% RSLogix 500 project Car Parking System Using Counters.RSS, saved by version 8.30.00.16 %
PROJECT "UNTITLED"    % processor: Bul.1763 MicroLogix 1100 Series B %

PROGRAM FILES
  LAD 2   6 rungs

DATA FILES
  O0 OUTPUT  4 elements
  I1 INPUT  6 elements
  S2 STATUS  66 elements
  B3 BINARY  1 elements
  T4 TIMER  1 elements
  C5 COUNTER  1 elements
  R6 CONTROL  1 elements
  N7 INTEGER  1 elements
  F8 FLOAT  1 elements

LADDER 2
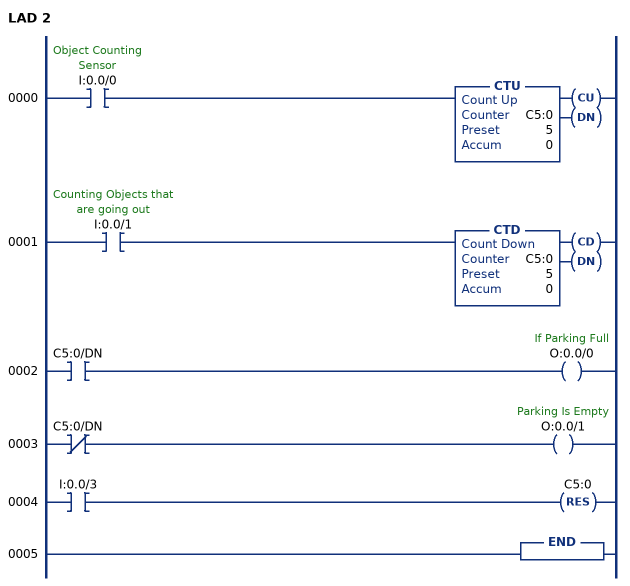
% Rung: 0 %
SOR XIC I:0.0/0 CTU C5:0 5 0 EOR
%   I:0.0/0  "Object Counting Sensor" %
% Rung: 1 %
SOR XIC I:0.0/1 CTD C5:0 5 0 EOR
%   I:0.0/1  "Counting Objects that are going out" %
% Rung: 2 %
SOR XIC C5:0/DN OTE O:0.0/0 EOR
%   O:0.0/0  "If Parking Full" %
% Rung: 3 %
SOR XIO C5:0/DN OTE O:0.0/1 EOR
%   O:0.0/1  "Parking Is Empty" %
% Rung: 4 %
SOR XIC I:0.0/3 RES C5:0 EOR
% Rung: 5 %
SOR END EOR

DATA TABLE (non-zero values as saved)
DATA C5
% .PRE .ACC %
% C5:0 % 5 0
